TYPE stError_AnalogueOutput :
STRUCT
	Out_Of_Range:BOOL;			//Input Value is outside range of Engineering Units
	Configuration_Error:BOOL;	//Engineering Units are not properly configured
END_STRUCT
END_TYPE

(* stored: Version 1.1.0.1, ProductVersion 3.1.4024.11
   DUT stError_AnalogueOutput: Id {cc192774-7426-4e7b-b022-46961ac77e78} *)
